FUNCTION_BLOCK FB_DLK
VAR_IN_OUT
	Parameter_init	: ST_DLK_Parameter;
END_VAR
VAR_OUTPUT
END_VAR
VAR
	{attribute 'OPC.UA.DA' := '1'}Zustand		: ST_DLK_Zustand;	
	{attribute 'OPC.UA.DA' := '1'}Parameter	: ST_DLK_Parameter;		
	Start_MK5	: TON;
	Zustandscheck	: FB_DLK_Zustandscheck;
END_VAR

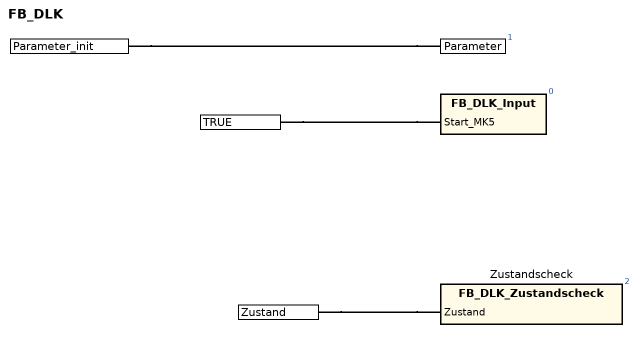
FB_DLK_Input(Start_MK5 := TRUE);
Parameter := Parameter_init;
Zustandscheck(Zustand := Zustand); // FB_DLK_Zustandscheck

END_FUNCTION_BLOCK

(* stored: Version 1.1.0.1, ProductVersion 3.1.4024.9
   POU FB_DLK: Id {acb81254-b358-4f61-ad15-2df99da36303}, SpecialFunc None *)
